(* PLC project PLC1, Beckhoff Automation GmbH TwinCAT PLC Control 3.5.21.30 *)
(* stored: creationDateTime 2026-05-11T22:43:57.9622111, modificationDateTime 2026-05-11T22:43:57.9622111 *)

FUNCTION F_ConsumeTime
VAR_INPUT
	Us		:UDINT;
END_VAR
VAR
		tCurr, tEnd : T_DCTIME64;
END_VAR

            tCurr := F_GetActualDcTime64();
tEnd  := tCurr + (Us * EC_DCTIME_TICKSPERMSEC64 / 1000);
WHILE (tCurr < tEnd) DO
	tCurr := F_GetActualDcTime64();
END_WHILE


          
END_FUNCTION
